(* IEC 61131-3 sources: Building-Automation/Water Treatment System/plc, 3 files *)

(* ---- desalination_controller.st ---- *)
// Desalination Controller Function Block
// Reverse Osmosis (RO) Process Control
// Author: PLC Control System
// Date: June 2025

FUNCTION_BLOCK DesalinationController
VAR_INPUT
    Enable          : BOOL := FALSE;    // Enable RO controller
    PressureSetpoint : REAL := 55.0;    // RO pressure setpoint (bar)
    RecoverySetpoint : REAL := 45.0;    // Recovery rate setpoint (%)
    Reset           : BOOL := FALSE;    // Reset controller
END_VAR

VAR_OUTPUT
    PumpSpeed       : REAL := 0.0;      // RO pump speed output (%)
    ConcentrateValve : REAL := 50.0;    // Concentrate valve position (%)
    SystemReady     : BOOL := FALSE;    // RO system ready
    SystemFault     : BOOL := FALSE;    // RO system fault
    CleaningRequired : BOOL := FALSE;   // Cleaning cycle required
END_VAR

VAR
    // PID controller for pressure
    PressurePID     : PID;
    PIDOutput       : REAL := 0.0;

    // Control parameters
    Kp              : REAL := 2.0;      // Proportional gain
    Ti              : REAL := 10.0;     // Integral time (s)
    Td              : REAL := 1.0;      // Derivative time (s)

    // Process variables
    PressureError   : REAL := 0.0;
    RecoveryRate    : REAL := 0.0;
    SaltRejection   : REAL := 0.0;

    // Fouling monitoring
    FoulingIndex    : REAL := 0.0;
    BaselinePressure : REAL := 55.0;
    PressureDrop    : REAL := 0.0;

    // Timers
    StartupTimer    : TON;
    StabilizeTimer  : TON;
    FaultTimer      : TON;

    // State machine
    ControlState    : INT := 0;

    // Operating hours for maintenance
    OperatingHours  : REAL := 0.0;
    CleaningCycles  : INT := 0;

END_VAR

// =====================================
// MAIN DESALINATION CONTROLLER
// =====================================

IF Reset THEN
    // Reset all controller states
    ControlState := 0;
    SystemFault := FALSE;
    PumpSpeed := 0.0;
    ConcentrateValve := 50.0;
    StartupTimer(IN := FALSE);
    StabilizeTimer(IN := FALSE);
    FaultTimer(IN := FALSE);
END_IF

IF Enable THEN
    // Update operating hours
    OperatingHours := OperatingHours + 0.001;  // Increment operating time

    // Calculate process variables
    CalculateProcessVariables();

    // RO system state machine
    CASE ControlState OF
        0: // Idle state
            PumpSpeed := 0.0;
            ConcentrateValve := 100.0;  // Fully open for startup
            SystemReady := FALSE;

            IF Enable AND NOT SystemFault THEN
                ControlState := 1;  // Move to startup
            END_IF

        1: // Startup sequence
            StartupTimer(IN := TRUE, PT := T#30s);

            // Gradual pump speed increase
            IF StartupTimer.ET < T#20s THEN
                PumpSpeed := REAL_TO_REAL(TIME_TO_DINT(StartupTimer.ET)) / 20000.0 * 40.0;  // Ramp to 40%
            ELSE
                PumpSpeed := 40.0;
            END_IF

            // Adjust concentrate valve during startup
            ConcentrateValve := 80.0;

            IF StartupTimer.Q THEN
                StartupTimer(IN := FALSE);
                ControlState := 2;  // Move to pressure control
            END_IF

        2: // Pressure control mode
            SystemReady := TRUE;

            // PID pressure control
            PressureError := PressureSetpoint - g_ROPressure;

            PressurePID(
                bEnable := TRUE,
                fSetpointValue := PressureSetpoint,
                fActualValue := g_ROPressure,
                fKp := Kp,
                fTn := Ti,
                fTv := Td,
                fOutMax := 90.0,
                fOutMin := 20.0
            );

            PumpSpeed := PressurePID.fOut;

            // Concentrate valve control for recovery optimization
            ControlConcentrateValve();

            // Monitor for faults
            MonitorSystemHealth();

            // Check for cleaning requirement
            CheckCleaningRequirement();

            IF SystemFault THEN
                ControlState := 3;  // Move to fault state
            END_IF

        3: // Fault state
            PumpSpeed := 0.0;
            ConcentrateValve := 100.0;
            SystemReady := FALSE;

            FaultTimer(IN := TRUE, PT := T#10s);
            IF FaultTimer.Q AND NOT SystemFault THEN
                FaultTimer(IN := FALSE);
                ControlState := 0;  // Return to idle
            END_IF
    END_CASE

ELSE
    // Controller disabled
    ControlState := 0;
    PumpSpeed := 0.0;
    ConcentrateValve := 100.0;
    SystemReady := FALSE;
    StartupTimer(IN := FALSE);
    StabilizeTimer(IN := FALSE);
    FaultTimer(IN := FALSE);
END_IF

// =====================================
// PROCESS CALCULATIONS
// =====================================
FUNCTION CalculateProcessVariables : BOOL
VAR_INPUT
END_VAR

    // Calculate recovery rate
    IF (g_PermeateFlow + g_ConcentrateFlow) > 0.0 THEN
        RecoveryRate := g_PermeateFlow / (g_PermeateFlow + g_ConcentrateFlow) * 100.0;
    ELSE
        RecoveryRate := 0.0;
    END_IF

    // Calculate salt rejection rate
    IF g_SeawaterQuality.TDS > 0.0 THEN
        SaltRejection := (1.0 - g_ProductQuality.TDS / g_SeawaterQuality.TDS) * 100.0;
    ELSE
        SaltRejection := 0.0;
    END_IF

    // Calculate fouling index
    PressureDrop := g_ROPressure - BaselinePressure;
    IF BaselinePressure > 0.0 THEN
        FoulingIndex := ABS(PressureDrop) / BaselinePressure * 100.0;
    END_IF

    // Update global RO status
    g_ROSystemData.Pressure := g_ROPressure;
    g_ROSystemData.Recovery := RecoveryRate;
    g_ROSystemData.Rejection := SaltRejection;
    g_ROSystemData.Permeate := g_PermeateFlow;
    g_ROSystemData.Concentrate := g_ConcentrateFlow;
    g_ROSystemData.Fouling := FoulingIndex;
    g_ROSystemData.CleanCycle := CleaningCycles;

    CalculateProcessVariables := TRUE;
END_FUNCTION

// =====================================
// CONCENTRATE VALVE CONTROL
// =====================================
FUNCTION ControlConcentrateValve : BOOL
VAR_INPUT
END_VAR
VAR
    RecoveryError   : REAL;
    ValveAdjustment : REAL;
END_VAR

    // Control concentrate valve to maintain recovery rate
    RecoveryError := RecoverySetpoint - RecoveryRate;

    // Adjust valve position based on recovery error
    IF ABS(RecoveryError) > 2.0 THEN  // Only adjust if error is significant
        ValveAdjustment := RecoveryError * 0.5;  // Gain factor

        ConcentrateValve := ConcentrateValve - ValveAdjustment;

        // Limit valve position
        IF ConcentrateValve > 90.0 THEN
            ConcentrateValve := 90.0;
        ELSIF ConcentrateValve < 30.0 THEN
            ConcentrateValve := 30.0;
        END_IF
    END_IF

    ControlConcentrateValve := TRUE;
END_FUNCTION

// =====================================
// SYSTEM HEALTH MONITORING
// =====================================
FUNCTION MonitorSystemHealth : BOOL
VAR_INPUT
END_VAR

    SystemFault := FALSE;

    // Check pressure limits
    IF g_ROPressure > 65.0 THEN  // Over pressure
        SystemFault := TRUE;
    END_IF

    IF g_ROPressure < 30.0 AND PumpSpeed > 50.0 THEN  // Pressure too low
        SystemFault := TRUE;
    END_IF

    // Check flow rates
    IF g_PermeateFlow < 50.0 AND PumpSpeed > 60.0 THEN  // Low permeate flow
        SystemFault := TRUE;
    END_IF

    // Check salt rejection
    IF SaltRejection < 95.0 THEN  // Poor salt rejection
        SystemFault := TRUE;
    END_IF

    // Check for membrane fouling
    IF FoulingIndex > 90.0 THEN  // Severe fouling
        SystemFault := TRUE;
    END_IF

    // Update global alarm status
    g_ROSystemAlarm := SystemFault;

    MonitorSystemHealth := TRUE;
END_FUNCTION

// =====================================
// CLEANING REQUIREMENT CHECK
// =====================================
FUNCTION CheckCleaningRequirement : BOOL
VAR_INPUT
END_VAR

    CleaningRequired := FALSE;

    // Check fouling level
    IF FoulingIndex > 70.0 THEN
        CleaningRequired := TRUE;
    END_IF

    // Check operating hours (monthly cleaning)
    IF OperatingHours > 720.0 THEN  // 30 days * 24 hours
        CleaningRequired := TRUE;
    END_IF

    // Check salt rejection degradation
    IF SaltRejection < 97.0 THEN
        CleaningRequired := TRUE;
    END_IF

    // Check recovery rate drop
    IF RecoveryRate < 40.0 THEN
        CleaningRequired := TRUE;
    END_IF

    CheckCleaningRequirement := TRUE;
END_FUNCTION

END_FUNCTION_BLOCK

// =====================================
// PID CONTROLLER FUNCTION BLOCK
// =====================================
FUNCTION_BLOCK PID
VAR_INPUT
    bEnable         : BOOL := FALSE;
    fSetpointValue  : REAL := 0.0;
    fActualValue    : REAL := 0.0;
    fKp             : REAL := 1.0;
    fTn             : REAL := 1.0;
    fTv             : REAL := 0.0;
    fOutMax         : REAL := 100.0;
    fOutMin         : REAL := 0.0;
    bReset          : BOOL := FALSE;
END_VAR

VAR_OUTPUT
    fOut            : REAL := 0.0;
    bARWActive      : BOOL := FALSE;
END_VAR

VAR
    fErrorOld       : REAL := 0.0;
    fIntegral       : REAL := 0.0;
    fDerivative     : REAL := 0.0;
    fError          : REAL := 0.0;
    fProportional   : REAL := 0.0;
    fPIDSum         : REAL := 0.0;
    fCycleTime      : REAL := 0.1;  // Assume 100ms cycle time
END_VAR

IF bReset THEN
    fIntegral := 0.0;
    fErrorOld := 0.0;
    fOut := 0.0;
    bARWActive := FALSE;
END_IF

IF bEnable THEN
    // Calculate error
    fError := fSetpointValue - fActualValue;

    // Proportional term
    fProportional := fKp * fError;

    // Integral term (if Tn > 0)
    IF fTn > 0.0 AND NOT bARWActive THEN
        fIntegral := fIntegral + (fKp * fError * fCycleTime / fTn);
    END_IF

    // Derivative term (if Tv > 0)
    IF fTv > 0.0 THEN
        fDerivative := fKp * fTv * (fError - fErrorOld) / fCycleTime;
    ELSE
        fDerivative := 0.0;
    END_IF

    // Sum PID terms
    fPIDSum := fProportional + fIntegral + fDerivative;

    // Apply output limits
    IF fPIDSum > fOutMax THEN
        fOut := fOutMax;
        bARWActive := TRUE;  // Anti-reset windup
    ELSIF fPIDSum < fOutMin THEN
        fOut := fOutMin;
        bARWActive := TRUE;  // Anti-reset windup
    ELSE
        fOut := fPIDSum;
        bARWActive := FALSE;
    END_IF

    // Store error for next cycle
    fErrorOld := fError;
ELSE
    fOut := 0.0;
    fIntegral := 0.0;
    fErrorOld := 0.0;
    bARWActive := FALSE;
END_IF

END_FUNCTION_BLOCK

(* ---- pump_controller.st ---- *)
// Pump Controller Function Block
// Multi-pump Control and Sequencing for Water Treatment System
// Author: PLC Control System
// Date: June 2025

FUNCTION_BLOCK PumpController
VAR_INPUT
    Enable          : BOOL := FALSE;    // Enable pump controller
    AutoMode        : BOOL := TRUE;     // Automatic mode selection
    ManualOverride  : BOOL := FALSE;    // Manual override mode
    Reset           : BOOL := FALSE;    // Reset controller
END_VAR

VAR_OUTPUT
    SystemReady     : BOOL := FALSE;    // Pump system ready
    SystemFault     : BOOL := FALSE;    // Pump system fault
    MaintenanceReq  : BOOL := FALSE;    // Maintenance required
END_VAR

VAR
    // Pump rotation and sequencing
    PumpRotationTimer   : TON;
    RotationInterval    : TIME := T#24h;    // 24-hour rotation
    ActivePumpIndex     : INT := 1;         // Currently active pump (1-4)
    PumpRunHours        : ARRAY[1..4] OF REAL; // Operating hours per pump

    // Pump control state machines
    IntakePumpState     : INT := 0;
    ROPumpState         : INT := 0;
    BoosterPump1State   : INT := 0;
    BoosterPump2State   : INT := 0;

    // Pump monitoring
    PumpStartDelay      : TON;
    PumpStopDelay       : TON;
    FaultCheckTimer     : TON;

    // Vibration and performance monitoring
    PerformanceCheck    : TON;
    PerformanceInterval : TIME := T#1h;

    // Pump efficiency tracking
    IntakeEfficiency    : REAL := 0.0;
    ROEfficiency        : REAL := 0.0;
    BoosterEfficiency1  : REAL := 0.0;
    BoosterEfficiency2  : REAL := 0.0;

END_VAR

// =====================================
// MAIN PUMP CONTROLLER
// =====================================

IF Reset THEN
    // Reset all pump states
    IntakePumpState := 0;
    ROPumpState := 0;
    BoosterPump1State := 0;
    BoosterPump2State := 0;
    SystemFault := FALSE;
    PumpRotationTimer(IN := FALSE);
    PumpStartDelay(IN := FALSE);
    PumpStopDelay(IN := FALSE);
END_IF

IF Enable THEN
    // Update pump operating hours
    UpdatePumpHours();

    // Pump rotation management
    ManagePumpRotation();

    // Individual pump controllers
    ControlIntakePump();
    ControlROPump();
    ControlBoosterPumps();

    // Monitor pump performance
    MonitorPumpPerformance();

    // Check maintenance requirements
    CheckMaintenanceRequirements();

    SystemReady := NOT SystemFault;

ELSE
    // Controller disabled - stop all pumps safely
    StopAllPumps();
    SystemReady := FALSE;
END_IF

// =====================================
// PUMP OPERATING HOURS TRACKING
// =====================================
FUNCTION UpdatePumpHours : BOOL
VAR_INPUT
END_VAR

    // Update operating hours for each pump
    IF g_IntakePump THEN
        PumpRunHours[1] := PumpRunHours[1] + 0.001;  // Increment time
        g_IntakePumpData.Hours := PumpRunHours[1];
    END_IF

    IF g_ROPump THEN
        PumpRunHours[2] := PumpRunHours[2] + 0.001;
        g_ROPumpData.Hours := PumpRunHours[2];
    END_IF

    IF g_BoosterPump1 THEN
        PumpRunHours[3] := PumpRunHours[3] + 0.001;
        g_BoosterPump1Data.Hours := PumpRunHours[3];
    END_IF

    IF g_BoosterPump2 THEN
        PumpRunHours[4] := PumpRunHours[4] + 0.001;
        g_BoosterPump2Data.Hours := PumpRunHours[4];
    END_IF

    UpdatePumpHours := TRUE;
END_FUNCTION

// =====================================
// PUMP ROTATION MANAGEMENT
// =====================================
FUNCTION ManagePumpRotation : BOOL
VAR_INPUT
END_VAR

    // Automatic pump rotation for equal wear
    PumpRotationTimer(IN := TRUE, PT := RotationInterval);

    IF PumpRotationTimer.Q AND AutoMode THEN
        PumpRotationTimer(IN := FALSE);

        // Rotate to next pump in sequence
        ActivePumpIndex := ActivePumpIndex + 1;
        IF ActivePumpIndex > 4 THEN
            ActivePumpIndex := 1;
        END_IF

        // Apply rotation logic for booster pumps
        RotateBoosterPumps();
    END_IF

    ManagePumpRotation := TRUE;
END_FUNCTION

FUNCTION RotateBoosterPumps : BOOL
VAR_INPUT
END_VAR

    // Rotate booster pumps based on operating hours
    IF PumpRunHours[3] > PumpRunHours[4] + 100.0 THEN
        // Pump 1 has significantly more hours, prefer pump 2
        IF g_BoosterPump1 AND NOT g_BoosterPump2 THEN
            g_BoosterPump1 := FALSE;
            PumpStopDelay(IN := TRUE, PT := T#5s);
            IF PumpStopDelay.Q THEN
                g_BoosterPump2 := TRUE;
                g_BoosterSpeed2 := g_BoosterSpeed1;
                g_BoosterSpeed1 := 0.0;
                PumpStopDelay(IN := FALSE);
            END_IF
        END_IF
    ELSIF PumpRunHours[4] > PumpRunHours[3] + 100.0 THEN
        // Pump 2 has significantly more hours, prefer pump 1
        IF g_BoosterPump2 AND NOT g_BoosterPump1 THEN
            g_BoosterPump2 := FALSE;
            PumpStopDelay(IN := TRUE, PT := T#5s);
            IF PumpStopDelay.Q THEN
                g_BoosterPump1 := TRUE;
                g_BoosterSpeed1 := g_BoosterSpeed2;
                g_BoosterSpeed2 := 0.0;
                PumpStopDelay(IN := FALSE);
            END_IF
        END_IF
    END_IF

    RotateBoosterPumps := TRUE;
END_FUNCTION

// =====================================
// INTAKE PUMP CONTROL
// =====================================
FUNCTION ControlIntakePump : BOOL
VAR_INPUT
END_VAR

    CASE IntakePumpState OF
        0: // Stopped
            g_IntakePump := FALSE;
            g_IntakePumpSpeed := 0.0;
            g_IntakePumpData.Running := FALSE;

            IF g_SystemRunning AND NOT SystemFault THEN
                IntakePumpState := 1;  // Start sequence
            END_IF

        1: // Starting
            PumpStartDelay(IN := TRUE, PT := T#3s);

            IF PumpStartDelay.Q THEN
                g_IntakePump := TRUE;
                g_IntakePumpSpeed := 30.0;  // Start at low speed
                PumpStartDelay(IN := FALSE);
                IntakePumpState := 2;  // Ramp up
            END_IF

        2: // Ramping up
            IF g_IntakePumpSpeed < g_IntakePumpSpeed THEN
                g_IntakePumpSpeed := g_IntakePumpSpeed + 5.0;
            ELSE
                IntakePumpState := 3;  // Normal operation
            END_IF

        3: // Normal operation
            g_IntakePumpData.Running := TRUE;

            // Monitor pump current and pressure
            MonitorIntakePump();

            IF NOT g_SystemRunning OR SystemFault THEN
                IntakePumpState := 4;  // Stop sequence
            END_IF

        4: // Stopping
            g_IntakePumpSpeed := g_IntakePumpSpeed - 10.0;

            IF g_IntakePumpSpeed <= 0.0 THEN
                g_IntakePump := FALSE;
                g_IntakePumpSpeed := 0.0;
                IntakePumpState := 0;  // Stopped
            END_IF
    END_CASE

    ControlIntakePump := TRUE;
END_FUNCTION

// =====================================
// RO PUMP CONTROL
// =====================================
FUNCTION ControlROPump : BOOL
VAR_INPUT
END_VAR

    CASE ROPumpState OF
        0: // Stopped
            g_ROPump := FALSE;
            g_ROPumpSpeed := 0.0;
            g_ROPumpData.Running := FALSE;

            IF g_SystemRunning AND NOT SystemFault AND g_IntakePump THEN
                ROPumpState := 1;  // Start sequence
            END_IF

        1: // Pre-start delay
            PumpStartDelay(IN := TRUE, PT := T#10s);

            IF PumpStartDelay.Q THEN
                g_ROPump := TRUE;
                g_ROPumpSpeed := 20.0;  // Start at very low speed
                PumpStartDelay(IN := FALSE);
                ROPumpState := 2;  // Gradual pressure build
            END_IF

        2: // Pressure building
            // Gradual speed increase to build pressure slowly
            IF g_ROPressure < 30.0 AND g_ROPumpSpeed < 50.0 THEN
                g_ROPumpSpeed := g_ROPumpSpeed + 2.0;  // Slow ramp
            ELSIF g_ROPressure >= 30.0 THEN
                ROPumpState := 3;  // Normal operation
            END_IF

            // Safety check - don't exceed pressure too quickly
            IF g_ROPressure > 40.0 THEN
                g_ROPumpSpeed := g_ROPumpSpeed - 5.0;
            END_IF

        3: // Normal operation
            g_ROPumpData.Running := TRUE;

            // Pump speed is controlled by desalination controller
            // Monitor pump performance here
            MonitorROPump();

            IF NOT g_SystemRunning OR SystemFault THEN
                ROPumpState := 4;  // Stop sequence
            END_IF

        4: // Stopping
            // Gradual pressure reduction
            g_ROPumpSpeed := g_ROPumpSpeed - 5.0;

            IF g_ROPumpSpeed <= 0.0 THEN
                g_ROPump := FALSE;
                g_ROPumpSpeed := 0.0;
                ROPumpState := 0;  // Stopped
            END_IF
    END_CASE

    ControlROPump := TRUE;
END_FUNCTION

// =====================================
// BOOSTER PUMPS CONTROL
// =====================================
FUNCTION ControlBoosterPumps : BOOL
VAR_INPUT
END_VAR

    // Booster Pump 1 Control
    CASE BoosterPump1State OF
        0: // Stopped
            g_BoosterPump1 := FALSE;
            g_BoosterSpeed1 := 0.0;
            g_BoosterPump1Data.Running := FALSE;

            IF g_RoofTank.Level < 70.0 AND g_GroundTank.Level > 30.0 THEN
                BoosterPump1State := 1;  // Start
            END_IF

        1: // Starting
            PumpStartDelay(IN := TRUE, PT := T#2s);

            IF PumpStartDelay.Q THEN
                g_BoosterPump1 := TRUE;
                g_BoosterSpeed1 := 40.0;  // Start speed
                PumpStartDelay(IN := FALSE);
                BoosterPump1State := 2;  // Running
            END_IF

        2: // Running
            g_BoosterPump1Data.Running := TRUE;

            // Speed control is handled by tank control logic
            MonitorBoosterPump1();

            IF g_RoofTank.Level > 90.0 OR g_GroundTank.Level < 20.0 THEN
                BoosterPump1State := 3;  // Stop
            END_IF

        3: // Stopping
            g_BoosterSpeed1 := g_BoosterSpeed1 - 10.0;

            IF g_BoosterSpeed1 <= 0.0 THEN
                g_BoosterPump1 := FALSE;
                g_BoosterSpeed1 := 0.0;
                BoosterPump1State := 0;  // Stopped
            END_IF
    END_CASE

    // Booster Pump 2 Control (similar logic with different conditions)
    CASE BoosterPump2State OF
        0: // Stopped
            g_BoosterPump2 := FALSE;
            g_BoosterSpeed2 := 0.0;
            g_BoosterPump2Data.Running := FALSE;

            // Start pump 2 if pump 1 is running and demand is high
            IF g_RoofTank.Level < 50.0 AND g_BoosterPump1 AND g_GroundTank.Level > 40.0 THEN
                BoosterPump2State := 1;  // Start
            END_IF

        1: // Starting
            PumpStartDelay(IN := TRUE, PT := T#2s);

            IF PumpStartDelay.Q THEN
                g_BoosterPump2 := TRUE;
                g_BoosterSpeed2 := 40.0;  // Start speed
                PumpStartDelay(IN := FALSE);
                BoosterPump2State := 2;  // Running
            END_IF

        2: // Running
            g_BoosterPump2Data.Running := TRUE;

            MonitorBoosterPump2();

            IF g_RoofTank.Level > 80.0 OR NOT g_BoosterPump1 THEN
                BoosterPump2State := 3;  // Stop
            END_IF

        3: // Stopping
            g_BoosterSpeed2 := g_BoosterSpeed2 - 10.0;

            IF g_BoosterSpeed2 <= 0.0 THEN
                g_BoosterPump2 := FALSE;
                g_BoosterSpeed2 := 0.0;
                BoosterPump2State := 0;  // Stopped
            END_IF
    END_CASE

    ControlBoosterPumps := TRUE;
END_FUNCTION

// =====================================
// PUMP MONITORING FUNCTIONS
// =====================================
FUNCTION MonitorIntakePump : BOOL
VAR_INPUT
END_VAR

    // Calculate pump efficiency (simplified)
    IF g_IntakePumpSpeed > 0.0 THEN
        IntakeEfficiency := (g_SeawaterQuality.FlowRate / g_IntakePumpSpeed) * 100.0;
    ELSE
        IntakeEfficiency := 0.0;
    END_IF

    // Update pump data structure
    g_IntakePumpData.Speed := g_IntakePumpSpeed;
    g_IntakePumpData.FlowRate := g_SeawaterQuality.FlowRate;
    g_IntakePumpData.Pressure := g_SeawaterQuality.Pressure;

    // Fault detection
    g_IntakePumpData.Fault := (g_IntakePumpData.Current > 15.0) OR  // Overcurrent
                             (IntakeEfficiency < 30.0 AND g_IntakePumpSpeed > 50.0);  // Low efficiency

    IF g_IntakePumpData.Fault THEN
        SystemFault := TRUE;
    END_IF

    MonitorIntakePump := TRUE;
END_FUNCTION

FUNCTION MonitorROPump : BOOL
VAR_INPUT
END_VAR

    // Calculate RO pump efficiency
    IF g_ROPumpSpeed > 0.0 THEN
        ROEfficiency := (g_ROPressure / g_ROPumpSpeed) * 100.0 / 55.0;  // Normalized to 55 bar
    ELSE
        ROEfficiency := 0.0;
    END_IF

    // Update pump data structure
    g_ROPumpData.Speed := g_ROPumpSpeed;
    g_ROPumpData.FlowRate := g_PermeateFlow;
    g_ROPumpData.Pressure := g_ROPressure;

    // Fault detection
    g_ROPumpData.Fault := (g_ROPumpData.Current > 25.0) OR  // Overcurrent
                         (g_ROPressure < 20.0 AND g_ROPumpSpeed > 60.0) OR  // Low pressure
                         (ROEfficiency < 40.0 AND g_ROPumpSpeed > 50.0);  // Low efficiency

    IF g_ROPumpData.Fault THEN
        SystemFault := TRUE;
    END_IF

    MonitorROPump := TRUE;
END_FUNCTION

FUNCTION MonitorBoosterPump1 : BOOL
VAR_INPUT
END_VAR

    // Calculate booster pump efficiency
    IF g_BoosterSpeed1 > 0.0 THEN
        BoosterEfficiency1 := (g_DistributionPressure / g_BoosterSpeed1) * 100.0 / 3.5;  // Normalized
    ELSE
        BoosterEfficiency1 := 0.0;
    END_IF

    // Update pump data structure
    g_BoosterPump1Data.Speed := g_BoosterSpeed1;
    g_BoosterPump1Data.Pressure := g_DistributionPressure;

    // Fault detection
    g_BoosterPump1Data.Fault := (g_BoosterPump1Data.Current > 12.0) OR  // Overcurrent
                               (BoosterEfficiency1 < 35.0 AND g_BoosterSpeed1 > 50.0);  // Low efficiency

    IF g_BoosterPump1Data.Fault THEN
        SystemFault := TRUE;
    END_IF

    MonitorBoosterPump1 := TRUE;
END_FUNCTION

FUNCTION MonitorBoosterPump2 : BOOL
VAR_INPUT
END_VAR

    // Calculate booster pump efficiency
    IF g_BoosterSpeed2 > 0.0 THEN
        BoosterEfficiency2 := (g_DistributionPressure / g_BoosterSpeed2) * 100.0 / 3.5;  // Normalized
    ELSE
        BoosterEfficiency2 := 0.0;
    END_IF

    // Update pump data structure
    g_BoosterPump2Data.Speed := g_BoosterSpeed2;
    g_BoosterPump2Data.Pressure := g_DistributionPressure;

    // Fault detection
    g_BoosterPump2Data.Fault := (g_BoosterPump2Data.Current > 12.0) OR  // Overcurrent
                               (BoosterEfficiency2 < 35.0 AND g_BoosterSpeed2 > 50.0);  // Low efficiency

    IF g_BoosterPump2Data.Fault THEN
        SystemFault := TRUE;
    END_IF

    MonitorBoosterPump2 := TRUE;
END_FUNCTION

// =====================================
// PERFORMANCE MONITORING
// =====================================
FUNCTION MonitorPumpPerformance : BOOL
VAR_INPUT
END_VAR

    PerformanceCheck(IN := TRUE, PT := PerformanceInterval);

    IF PerformanceCheck.Q THEN
        PerformanceCheck(IN := FALSE);

        // Log performance data and check trends
        // This would interface with data logging system

        // Check for performance degradation
        IF IntakeEfficiency < 40.0 THEN
            g_IntakePumpData.Maintenance := TRUE;
        END_IF

        IF ROEfficiency < 50.0 THEN
            g_ROPumpData.Maintenance := TRUE;
        END_IF

        IF BoosterEfficiency1 < 45.0 THEN
            g_BoosterPump1Data.Maintenance := TRUE;
        END_IF

        IF BoosterEfficiency2 < 45.0 THEN
            g_BoosterPump2Data.Maintenance := TRUE;
        END_IF
    END_IF

    MonitorPumpPerformance := TRUE;
END_FUNCTION

// =====================================
// MAINTENANCE REQUIREMENTS
// =====================================
FUNCTION CheckMaintenanceRequirements : BOOL
VAR_INPUT
END_VAR

    MaintenanceReq := FALSE;

    // Check operating hours for scheduled maintenance
    IF PumpRunHours[1] > 8760.0 THEN  // Annual maintenance
        g_IntakePumpData.Maintenance := TRUE;
        MaintenanceReq := TRUE;
    END_IF

    IF PumpRunHours[2] > 6000.0 THEN  // RO pump needs more frequent maintenance
        g_ROPumpData.Maintenance := TRUE;
        MaintenanceReq := TRUE;
    END_IF

    IF PumpRunHours[3] > 8760.0 THEN
        g_BoosterPump1Data.Maintenance := TRUE;
        MaintenanceReq := TRUE;
    END_IF

    IF PumpRunHours[4] > 8760.0 THEN
        g_BoosterPump2Data.Maintenance := TRUE;
        MaintenanceReq := TRUE;
    END_IF

    // Check for any pump faults
    IF g_IntakePumpData.Fault OR g_ROPumpData.Fault OR
       g_BoosterPump1Data.Fault OR g_BoosterPump2Data.Fault THEN
        MaintenanceReq := TRUE;
    END_IF

    CheckMaintenanceRequirements := TRUE;
END_FUNCTION

// =====================================
// EMERGENCY STOP ALL PUMPS
// =====================================
FUNCTION StopAllPumps : BOOL
VAR_INPUT
END_VAR

    // Immediate stop of all pumps
    g_IntakePump := FALSE;
    g_ROPump := FALSE;
    g_BoosterPump1 := FALSE;
    g_BoosterPump2 := FALSE;

    g_IntakePumpSpeed := 0.0;
    g_ROPumpSpeed := 0.0;
    g_BoosterSpeed1 := 0.0;
    g_BoosterSpeed2 := 0.0;

    // Reset all pump states
    IntakePumpState := 0;
    ROPumpState := 0;
    BoosterPump1State := 0;
    BoosterPump2State := 0;

    StopAllPumps := TRUE;
END_FUNCTION

END_FUNCTION_BLOCK

(* ---- main.st ---- *)
// Main Water Treatment System Control Program
// Seawater Desalination and Distribution System
// Author: PLC Control System
// Date: June 2025

PROGRAM Main
VAR
    // Local control variables
    StartupSequence     : INT := 0;         // Startup sequence step
    ShutdownSequence    : INT := 0;         // Shutdown sequence step
    ProductionCycle     : INT := 0;         // Production cycle step

    // Timer variables
    StartupTimer        : TON;              // System startup timer
    ShutdownTimer       : TON;              // System shutdown timer
    MaintenanceTimer    : TON;              // Maintenance interval timer
    ProductionTimer     : TON;              // Production cycle timer
    AlarmTimer          : TON;              // Alarm delay timer
    PumpRotationTimer   : TON;              // Pump rotation timer

    // Control flags
    SystemStartRequest  : BOOL := FALSE;    // System start request
    SystemStopRequest   : BOOL := FALSE;    // System stop request
    PumpRotationFlag    : BOOL := FALSE;    // Pump rotation flag
    CleaningCycleActive : BOOL := FALSE;    // RO cleaning cycle active

    // Process control variables
    RORecoveryRate      : REAL := 0.0;      // Calculated RO recovery rate
    SystemEfficiency    : REAL := 0.0;      // Overall system efficiency
    WaterLossRate       : REAL := 0.0;      // Water loss rate calculation

    // Maintenance tracking
    FilterHours         : ARRAY[1..5] OF REAL; // Filter operating hours
    PumpHours           : ARRAY[1..4] OF REAL; // Pump operating hours
    ROMembraneHours     : REAL := 0.0;      // RO membrane hours
    UVLampHours         : REAL := 0.0;      // UV lamp hours

END_VAR

// =====================================
// MAIN PROGRAM EXECUTION
// =====================================

// Read input signals and update system status
ReadInputs();

// Process emergency stop and safety systems
SafetyInterlocks();

// Handle system operating modes
CASE g_SystemMode OF
    STOPPED:
        SystemStoppedMode();

    STARTUP:
        SystemStartupMode();

    RUNNING:
        SystemRunningMode();

    SHUTDOWN:
        SystemShutdownMode();

    MAINTENANCE:
        MaintenanceMode();

    ALARM:
        AlarmMode();
END_CASE

// Execute water treatment processes
WaterTreatmentControl();

// Monitor and control water quality
WaterQualityControl();

// Tank level and distribution control
TankAndDistributionControl();

// Energy monitoring and optimization
EnergyManagement();

// Maintenance scheduling and alerts
MaintenanceManagement();

// Update outputs and HMI data
UpdateOutputs();

// =====================================
// INPUT PROCESSING
// =====================================
FUNCTION ReadInputs : BOOL
VAR_INPUT
END_VAR

    // Read digital inputs
    g_StartButton := StartButton;
    g_StopButton := StopButton;
    g_EmergencyButton := EmergencyButton;

    // Process start/stop requests
    IF g_StartButton AND NOT SystemStartRequest THEN
        SystemStartRequest := TRUE;
    END_IF

    IF g_StopButton AND NOT SystemStopRequest THEN
        SystemStopRequest := TRUE;
    END_IF

    // Update tank information
    g_GroundTank.Level := g_GroundTankLevel;
    g_GroundTank.Volume := g_GroundTank.Level * g_GroundTank.Capacity / 100.0;
    g_GroundTank.LowAlarm := g_GroundTankLevel < 20.0;
    g_GroundTank.HighAlarm := g_GroundTankLevel > 95.0;
    g_GroundTank.EmptyAlarm := g_GroundTankLevel < 5.0;

    g_RoofTank.Level := g_RoofTankLevel;
    g_RoofTank.Volume := g_RoofTank.Level * g_RoofTank.Capacity / 100.0;
    g_RoofTank.LowAlarm := g_RoofTankLevel < 30.0;
    g_RoofTank.HighAlarm := g_RoofTankLevel > 95.0;
    g_RoofTank.EmptyAlarm := g_RoofTankLevel < 10.0;

    // Update water quality data
    g_SeawaterQuality.TDS := g_SeawaterTDS;
    g_SeawaterQuality.Temperature := g_SeawaterTemp;
    g_ProductQuality.TDS := g_ProductTDS;
    g_ProductQuality.pH := g_ProductpH;
    g_ProductQuality.Turbidity := g_ProductTurbidity;
    g_ProductQuality.Chlorine := g_ChlorineLevel;
    g_ProductQuality.FlowRate := g_PermeateFlow;

    ReadInputs := TRUE;
END_FUNCTION

// =====================================
// SAFETY INTERLOCKS
// =====================================
FUNCTION SafetyInterlocks : BOOL
VAR_INPUT
END_VAR

    // Emergency stop processing
    IF g_EmergencyButton THEN
        g_EmergencyStop := TRUE;
        g_SystemMode := ALARM;

        // Stop all pumps immediately
        g_IntakePump := FALSE;
        g_PreFilterPump := FALSE;
        g_ROPump := FALSE;
        g_BoosterPump1 := FALSE;
        g_BoosterPump2 := FALSE;

        // Close critical valves
        g_IntakeValve := FALSE;
        g_ROPermeateValve := FALSE;

        g_SystemAlarm := TRUE;
        g_AlarmLight := TRUE;
    END_IF

    // Leak detection safety
    IF g_LeakDetector1 OR g_LeakDetector2 THEN
        g_LeakageAlarm := TRUE;

        // Stop pumps in affected zones
        IF g_LeakDetector1 THEN
            g_IntakePump := FALSE;
            g_PreFilterPump := FALSE;
        END_IF

        IF g_LeakDetector2 THEN
            g_ROPump := FALSE;
        END_IF
    END_IF

    // High pressure protection
    IF g_ROPressure > 65.0 THEN  // Emergency pressure limit
        g_ROPump := FALSE;
        g_ROSystemAlarm := TRUE;
        g_SystemAlarm := TRUE;
    END_IF

    // Tank overflow protection
    IF g_GroundTank.HighAlarm THEN
        g_IntakePump := FALSE;
        g_PreFilterPump := FALSE;
        g_ROPump := FALSE;
        g_GroundTankValve := FALSE;
    END_IF

    IF g_RoofTank.HighAlarm THEN
        g_BoosterPump1 := FALSE;
        g_BoosterPump2 := FALSE;
        g_RoofTankValve := FALSE;
    END_IF

    SafetyInterlocks := TRUE;
END_FUNCTION

// =====================================
// SYSTEM OPERATING MODES
// =====================================
FUNCTION SystemStoppedMode : BOOL
VAR_INPUT
END_VAR

    // All outputs off in stopped mode
    g_IntakePump := FALSE;
    g_PreFilterPump := FALSE;
    g_ROPump := FALSE;
    g_BoosterPump1 := FALSE;
    g_BoosterPump2 := FALSE;

    g_IntakeValve := FALSE;
    g_ROPermeateValve := FALSE;
    g_ConcentrateValve := FALSE;

    g_UVSterilizer := FALSE;
    g_ChlorineDosingPump := FALSE;
    g_pHDosingPump := FALSE;

    // Reset control variables
    StartupSequence := 0;
    ProductionCycle := 0;

    // Check for start request
    IF SystemStartRequest AND NOT g_EmergencyStop THEN
        g_SystemMode := STARTUP;
        SystemStartRequest := FALSE;
        g_StatusLight := TRUE;
    END_IF

    SystemStoppedMode := TRUE;
END_FUNCTION

FUNCTION SystemStartupMode : BOOL
VAR_INPUT
END_VAR

    // Startup sequence with proper delays
    CASE StartupSequence OF
        0: // Initialize startup
            StartupTimer(IN := TRUE, PT := T#2s);
            IF StartupTimer.Q THEN
                StartupTimer(IN := FALSE);
                StartupSequence := 1;
            END_IF

        1: // Open seawater intake valve
            g_IntakeValve := TRUE;
            StartupTimer(IN := TRUE, PT := T#5s);
            IF StartupTimer.Q THEN
                StartupTimer(IN := FALSE);
                StartupSequence := 2;
            END_IF

        2: // Start intake pump
            g_IntakePump := TRUE;
            g_IntakePumpSpeed := 60.0;  // Start at 60% speed
            StartupTimer(IN := TRUE, PT := T#10s);
            IF StartupTimer.Q THEN
                StartupTimer(IN := FALSE);
                StartupSequence := 3;
            END_IF

        3: // Start pre-filtration pump
            g_PreFilterPump := TRUE;
            StartupTimer(IN := TRUE, PT := T#15s);
            IF StartupTimer.Q THEN
                StartupTimer(IN := FALSE);
                StartupSequence := 4;
            END_IF

        4: // Start RO system
            g_ROPump := TRUE;
            g_ROPumpSpeed := 40.0;  // Start RO pump at low speed
            g_ConcentrateValve := TRUE;
            StartupTimer(IN := TRUE, PT := T#20s);
            IF StartupTimer.Q THEN
                StartupTimer(IN := FALSE);
                StartupSequence := 5;
            END_IF

        5: // Ramp up RO pressure gradually
            IF g_ROPressure < g_ROPressureSetpoint THEN
                g_ROPumpSpeed := g_ROPumpSpeed + 2.0;  // Increase speed gradually
                IF g_ROPumpSpeed > 90.0 THEN
                    g_ROPumpSpeed := 90.0;
                END_IF
            ELSE
                g_ROPermeateValve := TRUE;
                StartupSequence := 6;
            END_IF

        6: // Start post-treatment systems
            g_UVSterilizer := TRUE;
            g_GroundTankValve := TRUE;
            StartupTimer(IN := TRUE, PT := T#10s);
            IF StartupTimer.Q THEN
                StartupTimer(IN := FALSE);
                g_SystemMode := RUNNING;
                g_SystemRunning := TRUE;
                StartupSequence := 0;
            END_IF
    END_CASE

    // Abort startup on stop request or alarm
    IF SystemStopRequest OR g_EmergencyStop THEN
        g_SystemMode := SHUTDOWN;
        SystemStopRequest := FALSE;
        StartupSequence := 0;
    END_IF

    SystemStartupMode := TRUE;
END_FUNCTION

FUNCTION SystemRunningMode : BOOL
VAR_INPUT
END_VAR

    // Normal production operation
    g_SystemRunning := TRUE;
    g_StatusLight := TRUE;

    // Production cycle control
    CASE ProductionCycle OF
        0: // Normal production
            // Production is handled by other control functions
            ProductionTimer(IN := TRUE, PT := T#1h);  // 1 hour cycles
            IF ProductionTimer.Q THEN
                ProductionTimer(IN := FALSE);
                ProductionCycle := 1;  // Check for cleaning cycle
            END_IF

        1: // Check if RO cleaning needed
            IF g_ROSystemData.Fouling > 80.0 OR g_ROCleaningCycles < 1 THEN
                ProductionCycle := 2;  // Start cleaning cycle
                CleaningCycleActive := TRUE;
            ELSE
                ProductionCycle := 0;  // Continue production
            END_IF

        2: // RO cleaning cycle
            // Cleaning cycle implementation would go here
            // For now, simulate cleaning delay
            ProductionTimer(IN := TRUE, PT := T#30m);
            IF ProductionTimer.Q THEN
                ProductionTimer(IN := FALSE);
                g_ROCleaningCycles := g_ROCleaningCycles + 1;
                CleaningCycleActive := FALSE;
                ProductionCycle := 0;
            END_IF
    END_CASE

    // Check for stop request
    IF SystemStopRequest THEN
        g_SystemMode := SHUTDOWN;
        SystemStopRequest := FALSE;
    END_IF

    // Check for alarms that require shutdown
    IF g_EmergencyStop OR g_LeakageAlarm THEN
        g_SystemMode := ALARM;
    END_IF

    SystemRunningMode := TRUE;
END_FUNCTION

FUNCTION SystemShutdownMode : BOOL
VAR_INPUT
END_VAR

    // Controlled shutdown sequence
    CASE ShutdownSequence OF
        0: // Stop dosing pumps first
            g_ChlorineDosingPump := FALSE;
            g_pHDosingPump := FALSE;
            ShutdownTimer(IN := TRUE, PT := T#5s);
            IF ShutdownTimer.Q THEN
                ShutdownTimer(IN := FALSE);
                ShutdownSequence := 1;
            END_IF

        1: // Close permeate valve and reduce RO pressure
            g_ROPermeateValve := FALSE;
            g_ROPumpSpeed := g_ROPumpSpeed - 10.0;
            IF g_ROPumpSpeed <= 0.0 THEN
                g_ROPump := FALSE;
                ShutdownSequence := 2;
            END_IF

        2: // Stop RO pump and close concentrate valve
            g_ROPump := FALSE;
            g_ConcentrateValve := FALSE;
            ShutdownTimer(IN := TRUE, PT := T#10s);
            IF ShutdownTimer.Q THEN
                ShutdownTimer(IN := FALSE);
                ShutdownSequence := 3;
            END_IF

        3: // Stop pre-filtration pump
            g_PreFilterPump := FALSE;
            ShutdownTimer(IN := TRUE, PT := T#5s);
            IF ShutdownTimer.Q THEN
                ShutdownTimer(IN := FALSE);
                ShutdownSequence := 4;
            END_IF

        4: // Stop intake pump and close intake valve
            g_IntakePump := FALSE;
            g_IntakeValve := FALSE;
            ShutdownTimer(IN := TRUE, PT := T#10s);
            IF ShutdownTimer.Q THEN
                ShutdownTimer(IN := FALSE);
                ShutdownSequence := 5;
            END_IF

        5: // Stop remaining systems
            g_UVSterilizer := FALSE;
            g_GroundTankValve := FALSE;
            g_RoofTankValve := FALSE;
            g_SystemMode := STOPPED;
            g_SystemRunning := FALSE;
            g_StatusLight := FALSE;
            ShutdownSequence := 0;
    END_CASE

    SystemShutdownMode := TRUE;
END_FUNCTION

// =====================================
// WATER TREATMENT CONTROL
// =====================================
FUNCTION WaterTreatmentControl : BOOL
VAR_INPUT
END_VAR

    IF g_SystemRunning THEN
        // RO pressure control
        DesalinationController();

        // Water quality control
        WaterQualityController();

        // Pump control and sequencing
        PumpController();
    END_IF

    WaterTreatmentControl := TRUE;
END_FUNCTION

FUNCTION WaterQualityControl : BOOL
VAR_INPUT
END_VAR

    IF g_SystemRunning THEN
        // pH control
        IF g_ProductQuality.pH < g_ProductpHMin THEN
            g_pHDosingPump := TRUE;
            g_pHDoseRate := (g_ProductpHMin - g_ProductQuality.pH) * 20.0;
        ELSIF g_ProductQuality.pH > g_ProductpHMax THEN
            g_pHDosingPump := TRUE;
            g_pHDoseRate := (g_ProductQuality.pH - g_ProductpHMax) * 20.0;
        ELSE
            g_pHDosingPump := FALSE;
            g_pHDoseRate := 0.0;
        END_IF

        // Chlorine dosing control
        IF g_ProductQuality.Chlorine < g_ChlorineSetpoint THEN
            g_ChlorineDosingPump := TRUE;
            g_ChlorineRate := (g_ChlorineSetpoint - g_ProductQuality.Chlorine) * 50.0;
        ELSE
            g_ChlorineDosingPump := FALSE;
            g_ChlorineRate := 0.0;
        END_IF

        // Water quality alarms
        g_WaterQualityAlarm := (g_ProductQuality.TDS > g_ProductTDSLimit) OR
                              (g_ProductQuality.pH < g_ProductpHMin) OR
                              (g_ProductQuality.pH > g_ProductpHMax) OR
                              (g_ProductQuality.Turbidity > 1.0);
    END_IF

    WaterQualityControl := TRUE;
END_FUNCTION

FUNCTION TankAndDistributionControl : BOOL
VAR_INPUT
END_VAR

    // Ground tank control
    IF g_GroundTank.Level < 30.0 AND g_SystemRunning THEN
        // Increase production if tank is low
        g_IntakePumpSpeed := 80.0;
    ELSIF g_GroundTank.Level > 90.0 THEN
        // Reduce production if tank is nearly full
        g_IntakePumpSpeed := 40.0;
    ELSE
        g_IntakePumpSpeed := 60.0;  // Normal production rate
    END_IF

    // Roof tank filling control
    IF g_RoofTank.Level < 50.0 AND g_GroundTank.Level > 40.0 THEN
        g_BoosterPump1 := TRUE;
        g_RoofTankValve := TRUE;
        g_BoosterSpeed1 := 70.0;

        // Use second pump if level is very low
        IF g_RoofTank.Level < 30.0 THEN
            g_BoosterPump2 := TRUE;
            g_BoosterSpeed2 := 70.0;
        END_IF
    ELSIF g_RoofTank.Level > 90.0 THEN
        g_BoosterPump1 := FALSE;
        g_BoosterPump2 := FALSE;
        g_RoofTankValve := FALSE;
    END_IF

    // Distribution pressure control
    IF g_DistributionPressure < g_DistPressureSetpoint - 0.5 THEN
        // Increase pump speed to maintain pressure
        IF g_BoosterSpeed1 < 90.0 THEN
            g_BoosterSpeed1 := g_BoosterSpeed1 + 5.0;
        END_IF
        IF g_RoofTank.Level < 70.0 AND g_BoosterSpeed2 < 90.0 THEN
            g_BoosterPump2 := TRUE;
            g_BoosterSpeed2 := g_BoosterSpeed2 + 5.0;
        END_IF
    ELSIF g_DistributionPressure > g_DistPressureSetpoint + 0.5 THEN
        // Reduce pump speed if pressure is too high
        IF g_BoosterSpeed1 > 30.0 THEN
            g_BoosterSpeed1 := g_BoosterSpeed1 - 5.0;
        END_IF
        IF g_BoosterSpeed2 > 30.0 THEN
            g_BoosterSpeed2 := g_BoosterSpeed2 - 5.0;
        ELSIF g_BoosterSpeed2 <= 30.0 THEN
            g_BoosterPump2 := FALSE;
        END_IF
    END_IF

    TankAndDistributionControl := TRUE;
END_FUNCTION

FUNCTION EnergyManagement : BOOL
VAR_INPUT
END_VAR

    // Calculate total power consumption
    g_PowerConsumption := 0.0;

    // Add pump power consumption (estimated)
    IF g_IntakePump THEN
        g_PowerConsumption := g_PowerConsumption + (g_IntakePumpSpeed / 100.0) * 2.5;  // 2.5 kW max
    END_IF

    IF g_ROPump THEN
        g_PowerConsumption := g_PowerConsumption + (g_ROPumpSpeed / 100.0) * 7.5;  // 7.5 kW max
    END_IF

    IF g_BoosterPump1 THEN
        g_PowerConsumption := g_PowerConsumption + (g_BoosterSpeed1 / 100.0) * 3.0;  // 3.0 kW max
    END_IF

    IF g_BoosterPump2 THEN
        g_PowerConsumption := g_PowerConsumption + (g_BoosterSpeed2 / 100.0) * 3.0;  // 3.0 kW max
    END_IF

    // Add auxiliary equipment power
    IF g_UVSterilizer THEN
        g_PowerConsumption := g_PowerConsumption + 1.2;  // UV sterilizer
    END_IF

    // Calculate specific energy consumption
    IF g_ProductQuality.FlowRate > 0.0 THEN
        g_SpecificEnergy := g_PowerConsumption / (g_ProductQuality.FlowRate * 0.06);  // kWh/m³
    END_IF

    EnergyManagement := TRUE;
END_FUNCTION

FUNCTION MaintenanceManagement : BOOL
VAR_INPUT
END_VAR

    // Track operating hours for maintenance scheduling
    IF g_SystemRunning THEN
        // Update pump operating hours
        IF g_IntakePump THEN
            PumpHours[1] := PumpHours[1] + 0.001;  // Add time increment
        END_IF

        IF g_ROPump THEN
            PumpHours[2] := PumpHours[2] + 0.001;
            ROMembraneHours := ROMembraneHours + 0.001;
        END_IF

        IF g_BoosterPump1 THEN
            PumpHours[3] := PumpHours[3] + 0.001;
        END_IF

        IF g_BoosterPump2 THEN
            PumpHours[4] := PumpHours[4] + 0.001;
        END_IF

        IF g_UVSterilizer THEN
            UVLampHours := UVLampHours + 0.001;
        END_IF
    END_IF

    // Check maintenance intervals
    g_MaintenanceAlarm := (PumpHours[1] > 8760.0) OR  // Annual maintenance
                         (PumpHours[2] > 8760.0) OR
                         (PumpHours[3] > 8760.0) OR
                         (PumpHours[4] > 8760.0) OR
                         (ROMembraneHours > 17520.0) OR  // 2 years
                         (UVLampHours > 8760.0);  // Annual UV lamp replacement

    MaintenanceManagement := TRUE;
END_FUNCTION

FUNCTION AlarmMode : BOOL
VAR_INPUT
END_VAR

    // In alarm mode, maintain safe state
    g_SystemAlarm := TRUE;
    g_AlarmLight := TRUE;

    // Allow reset only if emergency stop is cleared and no active alarms
    IF NOT g_EmergencyStop AND NOT g_LeakageAlarm AND NOT g_WaterQualityAlarm THEN
        // Reset emergency stop if button is released
        IF NOT g_EmergencyButton THEN
            g_EmergencyStop := FALSE;
            g_SystemMode := STOPPED;
            g_SystemAlarm := FALSE;
            g_AlarmLight := FALSE;
        END_IF
    END_IF

    AlarmMode := TRUE;
END_FUNCTION

FUNCTION UpdateOutputs : BOOL
VAR_INPUT
END_VAR

    // Update all output signals based on control logic
    // Digital outputs are already set by control functions

    // Update analog outputs
    IntakePumpSpeed := g_IntakePumpSpeed;
    ROPumpSpeed := g_ROPumpSpeed;
    BoosterSpeed1 := g_BoosterSpeed1;
    BoosterSpeed2 := g_BoosterSpeed2;
    ChlorineRate := g_ChlorineRate;
    pHDoseRate := g_pHDoseRate;

    // Update status indicators
    StatusLight := g_StatusLight;
    AlarmLight := g_AlarmLight;
    SystemAlarm := g_SystemAlarm;

    UpdateOutputs := TRUE;
END_FUNCTION

END_PROGRAM
